FUNCTION F_UpdateEventTimeStampWithSystemTime 
VAR_INPUT
	stEvent : REFERENCE TO St_Event ;
END_VAR
VAR
	fbGETSYSTEMTIME : GETSYSTEMTIME ;
	
	stFileTime : T_FILETIME ;
	
END_VAR

fbGETSYSTEMTIME (timeLoDW => stFileTime.dwLowDateTime,
				 timeHiDW => stFileTime.dwHighDateTime) ;
				 
stEvent.dtTimeStamp := FILETIME_TO_DT(fileTime := stFileTime ) ;

END_FUNCTION

(* stored: Version 1.1.0.1, ProductVersion 3.1.4024.12
   POU F_UpdateEventTimeStampWithSystemTime: Id {6e15ab70-44aa-44fe-86f0-070b91b3947a}, SpecialFunc None *)
